FUNCTION_BLOCK fAI
VAR_INPUT
	iAnalog: INT;
	///Valor minino del sensor en UF
	iPFSnsMinUF: INT:= 0;
	///Valor maxino del sensor en UF
	iPFSnsMaxUF: INT:= 32767;
	iPF_Ana_min: INT := 0;
	iPF_Ana_max: INT := 100;
END_VAR
VAR_OUTPUT
	rValor: REAL;
	rAnaUF: REAL;
END_VAR
VAR
	rAna_min: REAL := 0;
	rAna_max: REAL := 32767;
	bCre: BOOL;
	rSns_min: REAL;
	rSns_max: REAL;
	rReadAna: REAL;
	rSns_min_UF: REAL;
	rSns_max_UF: REAL;
END_VAR

(*-------------------------------------------------------------------------------------------------------*)

	(*Comprobar lectura creciente o decreciente*)
IF iPF_Ana_min > iPF_Ana_max THEN
		bCre:=TRUE; 
		ELSE
		bCre:=FALSE;
END_IF


	(*valores min y maximo de la analogica*)
IF bCre 
	THEN
		rAna_min:=((INT_TO_REAL(iPF_Ana_min)/100.0)*32767);
		rAna_max:=((INT_TO_REAL(iPF_Ana_max)/100.0)*32767);
	ELSE
		rAna_max:=((INT_TO_REAL(iPF_Ana_min)/100.0)*32767);
		rAna_min:=((INT_TO_REAL(iPF_Ana_max)/100.0)*32767);
END_IF
	(*salidas porentual nivel*)
	rSns_min_UF:=INT_TO_REAL(iPFSnsMinUF);
	rSns_max_UF:=INT_TO_REAL(iPFSnsMaxUF);
	(*Buscar valor de lectrua analogico*)
	rReadAna:=rValor;					(*FALTA REVISAR DIRECCION HARD*)
	(*Carregar lectura percentual *)
	rValor:=Canvi_Escala(
			In:= rReadAna, 
			In_Min:= rAna_min, 
			In_Max:= rAna_max, 
			Out_Min:= 0, 
			Out_Max:= 100);
	(*Carregar lectura Analog UF*)
	rAnaUF:=Canvi_Escala(
			In:= rReadAna, 
			In_Min:= 0, 
			In_Max:= 32767, 
			Out_Min:= rSns_min, 
			Out_Max:= rSns_max);

END_FUNCTION_BLOCK

(* stored: Version 1.1.0.1, ProductVersion 3.1.4024.10
   POU fAI: Id {99df198b-20b0-40cc-b0d0-936c59e41b00}, SpecialFunc None *)
